// LS Electric XG5000 project: 기본회로1
// 240116 12:30
// PLC LSPLC

PROGRAM NewProgram (task: 스캔 프로그램)

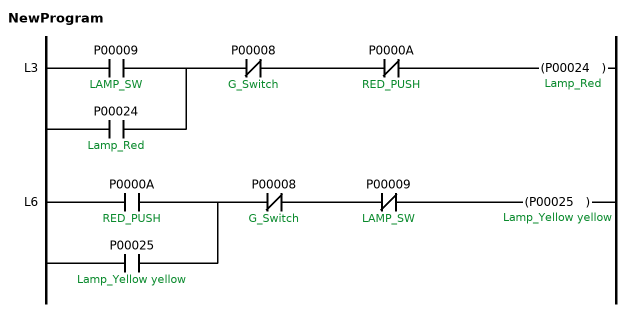
; L3
LOAD      P00009	// LAMP_SW
OR        P00024	// Lamp_Red
AND NOT   P00008	// G_Switch
AND NOT   P0000A	// RED_PUSH
OUT       P00024	// Lamp_Red
; L6
LOAD      P0000A	// RED_PUSH
OR        P00025	// Lamp_Yellow yellow
AND NOT   P00008	// G_Switch
AND NOT   P00009	// LAMP_SW
OUT       P00025	// Lamp_Yellow yellow

VARIABLES AND COMMENTS (devices not used above)
P00026	BIT	Lamp_Green // Lamp_green
P0000B	BIT	Swich_b // swich_b
P0000C	BIT	swich_c